(* PLC project TC3_TE1400_GeneratedModule_TempContr_FB, Beckhoff Automation GmbH TwinCAT 3 Function - TE1400 1.1.1105 *)
(* stored: companyURL www.beckhoff.com, creationDateTime 2013-10-01T13:17:51 *)

FUNCTION_BLOCK FB_TempContr
  VAR_INPUT
    ObjectID : OTCID;  (* object ID of the simulink module instance to be called *)
    stInputs : ExtU_TempContr_T;  (* input structure (also accessible via property 'Inputs') *)
  END_VAR
  VAR_OUTPUT
    hResult : HRESULT;  (* hResult of interface calls (0 if no error) *)
    iidFailedInterface : IID;  (* interface ID of the failing interface if hResult <> 0 *)
    bReady : BOOL;  (* TRUE, if initialized successfully *)
    stOutputs : ExtY_TempContr_T;  (* output structure (also accessible via property 'Outputs') *)
  END_VAR
  VAR
    ipObjSrv : ITComObjectServer;  (* Interface pointer to the Object Server *)
    ipTcCyclic : ITcCyclic;  (* Interface pointers to the used interfaces *)
    ipTcPostCyclic : ITcPostCyclic;
    ipTcAdi : ITcADI;
    pInputs : POINTER TO ExtU_TempContr_T;  (* pointer to the input process image of the simulink module *)
    pOutputs : POINTER TO ExtY_TempContr_T;  (* pointer to the output process image of the simulink module *)
  END_VAR

            
          

METHOD FB_EXIT : BOOL
  VAR_INPUT
    bInCopyCode : BOOL;  (* bei TRUE wird die exit-Methode aufgerufen, um die Instanz zu verlassen, die hinterher kopiert wird (Online Change). *)
  END_VAR
                  
// release ADI interface pointer
IF (ipTcAdi<>0) THEN
  ipTcAdi.TcRelease();
  ipTcAdi := 0;
END_IF

// release other interface pointers
IF (ipTcCyclic<>0) THEN
  ipTcCyclic.TcRelease();
  ipTcCyclic := 0;
END_IF
IF (ipTcPostCyclic<>0) THEN
  ipTcPostCyclic.TcRelease();
  ipTcPostCyclic := 0;
END_IF
IF (ipObjSrv<>0) THEN
ipObjSrv.TcRelease();
  ipObjSrv := 0;
END_IF
                  
                
END_METHOD

METHOD FB_INIT : BOOL
  VAR_INPUT
    bInitRetains : BOOL;
    bInCopyCode : BOOL;
    oid : OTCID;
  END_VAR
                  
hResult := S_OK;

// set object ID, if defined in the argument list
if(oid>0) THEN
 ObjectID := oid;
END_IF

// get object server
hResult := FW_ObjMgr_GetObjectServer(_AppInfo.ObjId,ADR(ipObjSrv));
IF (hResult<>S_OK) THEN
 iidFailedInterface := IID_ITComObjectServer;
END_IF


//get interface pointer to the cyclic interface of the simulink module
IF (hResult=S_OK) THEN
 hResult := ipObjSrv.TcQueryObjectInterface(oid:= ObjectID, iid:= IID_ITCCYCLIC, pipItf:=ADR(ipTcCyclic));
 IF (hResult<>S_OK) THEN
  iidFailedInterface := IID_ITCCYCLIC;
 END_IF
END_IF

//get interface pointer to the cyclic interface of the simulink module
IF (hResult=S_OK) THEN
 hResult := ipObjSrv.TcQueryObjectInterface(oid:= ObjectID, iid:= IID_ITCPOSTCYCLIC, pipItf:=ADR(ipTcPostCyclic));
 IF (hResult<>S_OK) THEN
  iidFailedInterface := IID_ITCPOSTCYCLIC;
 END_IF
END_IF

//get interface pointer to the adi interface of the simulink module
IF (hResult=S_OK) THEN
 hResult := ipObjSrv.TcQueryObjectInterface(oid:= ObjectID, iid:= IID_ITcADI, pipItf:=ADR(ipTcAdi));
 IF (hResult<>S_OK) THEN
  iidFailedInterface := IID_ITcADI;
 END_IF
END_IF

// check state
bReady := (hResult=S_OK);

// free pointer if not ready
IF NOT bReady THEN
  FB_EXIT(false);
END_IF

// return value
FB_INIT := (hResult=S_OK);    
                  
                
END_METHOD

METHOD FB_EXECUTE
                  
IF NOT bReady THEN
RETURN;
END_IF

// get pointer to the input process image
IF (hResult=S_OK) THEN
  hResult := ipTcAdi.GetImagePtr(size:= SIZEOF(ExtU_TempContr_T) , offs:=0 , adi_x:=0 , ppData:=ADR(pInputs));
  IF (hResult<>S_OK) THEN
    iidFailedInterface := IID_ITcADI;
  END_IF
END_IF

// get pointer to the output process image
IF (hResult=S_OK) THEN
  hResult := ipTcAdi.GetImagePtr(size:= SIZEOF(ExtY_TempContr_T) , offs:=0 , adi_x:=1 , ppData:=ADR(pOutputs));
  IF (hResult<>S_OK) THEN
    iidFailedInterface := IID_ITcADI;
  END_IF
END_IF


// copy inputs
IF (pInputs<>0) THEN
  pInputs^ := stInputs;
END_IF

// call output update
IF (ipTcCyclic<>0) THEN
  hResult := ipTcCyclic.CycleUpdate(ipTask:= 0, ipCaller:= 0, context:= 0);
ELSE
  hResult := 1;
END_IF

// copy outputs
IF (pOutputs<>0) THEN
  stOutputs := pOutputs^;
END_IF

// call state update
IF (ipTcPostCyclic<>0) THEN
  hResult := ipTcPostCyclic.PostCyclicUpdate(ipTask:= 0, ipCaller:= 0, context:= 0);
ELSE
  hResult := 1;
END_IF

// release process image pointers
  IF (pInputs<>0) THEN
    ipTcAdi.ReleaseImagePtr(pData:=pInputs);
    pInputs := 0;
  END_IF
  IF (pOutputs<>0) THEN
    ipTcAdi.ReleaseImagePtr(pData:=pOutputs);
    pOutputs := 0;
  END_IF
                  
                
END_METHOD
END_FUNCTION_BLOCK
